TYPE HMIXTSHelper_typ :
STRUCT
	Mover	: ARRAY[0..GVL.NUM_MOVERS-1] OF HMIXTSMoverHelper_typ;
END_STRUCT
END_TYPE

(* stored: Version 1.1.0.1, ProductVersion 3.1.4024.12
   DUT HMIXTSHelper_typ: Id {c8a0cee8-4307-0271-148b-b2649db85418} *)
